# B&R Automation Studio project Tuerschleuse_BR
Automation Studio 4.7.2.98

## Configuration Config1

CPU X20CP1584, AutomationRuntime A4.73, Build 4.1.2, Vc V4.72.0

### Hardware
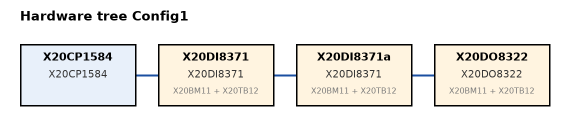
```
X20BM11 : X20BM11 v1.0.0.1  [X2X1 -> X20CP1584.IF6]
X20BM11a : X20BM11 v1.0.0.1  [X2X1 -> X20BM11.X2X2]
X20BM11b : X20BM11 v1.0.0.1  [X2X1 -> X20BM11a.X2X2]
X20CP1584 : X20CP1584 v1.6.0.0
  Connector IF2:
    ActivateDevice = 1
    Mode = Manual
    InternetAddress = 10.36.37.18
    SubnetMask = 255.255.255.0
  ConfigurationID = Door_control_Config1
X20DI8371 : X20DI8371 v1.0.2.0  [SS1 -> X20TB12.SS; SL -> X20BM11.SL1]
X20DI8371a : X20DI8371 v1.0.2.0  [SS1 -> X20TB12a.SS; SL -> X20BM11a.SL1]
X20DO8322 : X20DO8322 v1.1.0.0  [SS1 -> X20TB12b.SS; SL -> X20BM11b.SL1]
X20TB12 : X20TB12 v1.0.0.0
X20TB12a : X20TB12 v1.0.0.0
X20TB12b : X20TB12 v1.0.0.0
```

### IoMap.iom - X20CP1584/IoMap.iom
```iecst
VAR_CONFIG
	::S1 AT %IX."X20DI8371".DigitalInput01;
	::S2 AT %IX."X20DI8371".DigitalInput02;
	::S3 AT %IX."X20DI8371".DigitalInput03;
	::S4 AT %IX."X20DI8371".DigitalInput04;
	::S5 AT %IX."X20DI8371".DigitalInput05;
	::S6 AT %IX."X20DI8371".DigitalInput06;
	::S7 AT %IX."X20DI8371".DigitalInput07;
	::S8 AT %IX."X20DI8371".DigitalInput08;
	::B1 AT %IX."X20DI8371a".DigitalInput01 INVERSE;
	::B2 AT %IX."X20DI8371a".DigitalInput02 INVERSE;
	::M1L  AT %QX."X20DO8322".DigitalOutput02;
	::M2R  AT %QX."X20DO8322".DigitalOutput03;
	::M2L  AT %QX."X20DO8322".DigitalOutput04;
	::Anzeige_1 AT %QX."X20DO8322".DigitalOutput05;
	::Anzeige_2  AT %QX."X20DO8322".DigitalOutput06;
	::M1R AT %QX."X20DO8322".DigitalOutput01;
END_VAR
```

## Logical view

### Global.var - Global variables
```iecst
(*Eingänge*)
VAR
	S1 : BOOL;
	S2 : BOOL;
	S3 : BOOL;
	S4 : BOOL;
	S5 : BOOL;
	S6 : BOOL;
	S7 : BOOL;
	S8 : BOOL;
	B1 : BOOL;
	B2 : BOOL;
END_VAR
(*Ausgänge*)
VAR
	M1R : BOOL;
	M1L : BOOL;
	M2R : BOOL;
	M2L : BOOL;
	Anzeige_1 : BOOL;
	Anzeige_2 : BOOL;
END_VAR
```

### Program Logical/Program (ANSIC)

#### Cyclic.c
```c
#include <bur/plctypes.h>
#include <standard.h>

#ifdef _DEFAULT_INCLUDES
#include <AsDefault.h>
#endif

#define T_OPENED_DOOR 5000

struct motorDATA
{
	char M_rechts, M_links, stop_rechts, stop_links, lichtschranke, anzeige;
};

enum
{
	INIT, STOP, OPENS, OPENED, CLOSES, ERROR
};

char handleDoor(char state, struct motorDATA *motor, char s_open, char isOTHERdoorClosed, TON_typ *errorTimer);

void _CYCLIC ProgramCyclic(void)
{
	static TON_typ errorTimer_1, errorTimer_2;
	static struct motorDATA motorDATA_1={0,0,0,0,0}, motorDATA_2={0,0,0,0,0};
	static int state1, state2;

	errorTimer_1.PT = 8000;
	errorTimer_2.PT = 8000;

	motorDATA_1.lichtschranke = B1;
	motorDATA_1.stop_links = S5;
	motorDATA_1.stop_rechts = S6;

	motorDATA_2.lichtschranke = B2;
	motorDATA_2.stop_links = S7;
	motorDATA_2.stop_rechts = S8;

	state1 = handleDoor(state1, &motorDATA_1, (S1 | S3), S7, &errorTimer_1);
	state2 = handleDoor(state2, &motorDATA_2, (S4 | S2), S5, &errorTimer_2);

	M1R = motorDATA_1.M_rechts;
	M1L = motorDATA_1.M_links;
	Anzeige_1 = motorDATA_1.anzeige;

	M2R = motorDATA_2.M_rechts;
	M2L = motorDATA_2.M_links;
	Anzeige_2 = motorDATA_2.anzeige;
	TON(&errorTimer_1);
	TON(&errorTimer_2);

}

char handleDoor(char state, struct motorDATA *motor, char s_open, char isOTHERdoorClosed, TON_typ *errorTimer)
{
	static TON_typ doorOpenTimer, blinkTimer;
	doorOpenTimer.PT = 5000;
	blinkTimer.PT = 200;

	switch(state)
	{
		case INIT:
			motor->anzeige = 0;

			if(!motor->stop_links)
				state = CLOSES;
			if(motor->stop_links)
				state = STOP;
			break;

		case STOP:
			motor->M_rechts = 0;
			motor->M_links = 0;
			motor->anzeige = 0;

			if(s_open && isOTHERdoorClosed)
				state = OPENS;
			break;

		case OPENS:
			motor->M_rechts = 1;
			motor->M_links = 0;
			motor->anzeige = 0;

			if(motor->stop_rechts)
				state = OPENED;
			break;

		case OPENED:
			motor->M_rechts = 0;
			motor->M_links = 0;
			motor->anzeige = 0;
			doorOpenTimer.IN = 1;

			if(doorOpenTimer.Q)
			{
				doorOpenTimer.IN = 0;
				state = CLOSES;
			}
			break;

		case CLOSES:
			motor->M_rechts = 0;
			motor->M_links = 1;

			blinkTimer.IN = 1;
			if(blinkTimer.Q)
			{
				blinkTimer.IN = 0;
				//Toggle anzeigeLED
				motor->anzeige ^= 1;
			}

			if(motor->stop_links)
				state = STOP;
			if(motor->lichtschranke)
				state = OPENS;
			if(s_open)
				state = OPENS;

			break;

		case ERROR:
			motor->M_rechts = 0;
			motor->M_links = 0;
			motor->anzeige = 1;

			if(s_open)
				state = CLOSES;
			break;
	}
	//errrorHandling
	errorTimer->IN = ((motor->M_links) || (motor->M_rechts));

	if(errorTimer->Q)
		state = ERROR;

	TON(&doorOpenTimer);
	TON(&blinkTimer);

	return state;
}
```

Listed in the project but not available here: Logical/Global.typ, Logical/Libraries
